// TIA Portal V20 export
DATA_BLOCK "InstCallEquipment"   // DB136
{ DB_Accessible_From_OPC_UA := 'FALSE' }
AUTHOR : ERsystem_FA2_DH. Kim
// stored: AssignedProDiagFB Unit1.Em2.ProDiag, DBAccessibleFromOPCUA false, DBAccessibleFromWebserver false, InstanceOfName Unit1.Em2.CallEquipment, InstanceOfType FB, Namespace Unit1.Em2
"Unit1.Em2.CallEquipment"
   // VAR_INPUT
   //    ZoneOperationEnable { ExternalWritable := 'False'} : "LWONIK_typeSafetyZoneManualOperation";
   // END_VAR
   // VAR_IN_OUT
   //    unitStatus : "LAF_typeUnitStatus";
   //    unitAlarmDB : "LAF_typeAlarms";
   //    emFeedback : "LUC_typeEmFeedback";
   // END_VAR
   // VAR
   //    instSequenceSemiAutoSplice { ExternalWritable := 'False'} : "Unit1.Em2.Sequence_1_SemiAutoSplice";
   //    instHomeJob1 { S7_SetPoint := 'True'} : "LAF_SelectJob";
   //    instJob2 { S7_SetPoint := 'True'} : "LAF_SelectJob";
   //    instJob3 { S7_SetPoint := 'True'} : "LAF_SelectJob";
   //    instJob4 { S7_SetPoint := 'True'} : "LAF_SelectJob";
   //    instJob5 { S7_SetPoint := 'True'} : "LAF_SelectJob";
   //    instJob6 { S7_SetPoint := 'True'} : "LAF_SelectJob";
   //    instJob7 { S7_SetPoint := 'True'} : "LAF_SelectJob";
   //    instJob8 { S7_SetPoint := 'True'} : "LAF_SelectJob";
   //    instJob9 { S7_SetPoint := 'True'} : "LAF_SelectJob";
   //    instJob10 { S7_SetPoint := 'True'} : "LAF_SelectJob";
   //    instJob11 { S7_SetPoint := 'True'} : "LAF_SelectJob";
   //    instJob12 { S7_SetPoint := 'True'} : "LAF_SelectJob";
   //    instJob13 { S7_SetPoint := 'True'} : "LAF_SelectJob";
   //    instJob14 { S7_SetPoint := 'True'} : "LAF_SelectJob";
   //    instJob15 { S7_SetPoint := 'True'} : "LAF_SelectJob";
   //    instJob16 { S7_SetPoint := 'True'} : "LAF_SelectJob";
   //    instJob17 { S7_SetPoint := 'True'} : "LAF_SelectJob";
   //    instJob18 { S7_SetPoint := 'True'} : "LAF_SelectJob";
   //    instJob19 { S7_SetPoint := 'True'} : "LAF_SelectJob";
   //    instJob20 { S7_SetPoint := 'True'} : "LAF_SelectJob";
   //    instJob21 { S7_SetPoint := 'True'} : "LAF_SelectJob";
   //    instJob22 { S7_SetPoint := 'True'} : "LAF_SelectJob";
   //    instJob23 { S7_SetPoint := 'True'} : "LAF_SelectJob";
   //    instJob24 { S7_SetPoint := 'True'} : "LAF_SelectJob";
   //    instJob25 { S7_SetPoint := 'True'} : "LAF_SelectJob";
   //    instJob26 { S7_SetPoint := 'True'} : "LAF_SelectJob";
   //    instJob27 { S7_SetPoint := 'True'} : "LAF_SelectJob";
   //    instJob28 { S7_SetPoint := 'True'} : "LAF_SelectJob";
   //    instJob29 { S7_SetPoint := 'True'} : "LAF_SelectJob";
   //    instJob30 { S7_SetPoint := 'True'} : "LAF_SelectJob";
   //    instBtmSepaVaccumJob4 { S7_SetPoint := 'True'} : "LAF_SelectJob";
   //    instCuttingJob5 { S7_SetPoint := 'True'} : "LAF_SelectJob";
   //    instTopSepaTransferJob6 { S7_SetPoint := 'True'} : "LAF_SelectJob";
   //    instBtmSepaTransferJob7 { S7_SetPoint := 'True'} : "LAF_SelectJob";
   //    instSuctionPadDownJob8 { S7_SetPoint := 'True'} : "LAF_SelectJob";
   //    instTopSepaReMoveJob9 { S7_SetPoint := 'True'} : "LAF_SelectJob";
   //    instBtmSepaReMoveJob10 { S7_SetPoint := 'True'} : "LAF_SelectJob";
   //    instTopSpliceRoateJob11 { S7_SetPoint := 'True'} : "LAF_SelectJob";
   //    instBtmSpliceRoateJob12 { S7_SetPoint := 'True'} : "LAF_SelectJob";
   //    instTopTapingStartJob13 { S7_SetPoint := 'True'} : "LAF_SelectJob";
   //    instBtmTapingStartJob14 { S7_SetPoint := 'True'} : "LAF_SelectJob";
   //    instTapingFinishJob15 { S7_SetPoint := 'True'} : "LAF_SelectJob";
   //    instFullAutoSplicingJob30 { S7_SetPoint := 'True'} : "LAF_SelectJob";
   //    instIsLink { S7_SetPoint := 'True'} : "LAF_SelectJob";
   //    instcmSuctionPadTopUpDown { ExternalAccessible := 'False'; ExternalVisible := 'False'; ExternalWritable := 'False'; S7_SetPoint := 'True'} : "LBC_TwoWayActuatorCn";
   //    instcmSuctionPadBtmUpDown { ExternalAccessible := 'False'; ExternalVisible := 'False'; ExternalWritable := 'False'; S7_SetPoint := 'True'} : "LBC_TwoWayActuatorCn";
   //    instcmCutterUpDown { ExternalAccessible := 'False'; ExternalVisible := 'False'; ExternalWritable := 'False'; S7_SetPoint := 'True'} : "LBC_TwoWayActuatorCn";
   //    instcmTapeTopUpDown { ExternalAccessible := 'False'; ExternalVisible := 'False'; ExternalWritable := 'False'; S7_SetPoint := 'True'} : "LBC_TwoWayActuatorCn";
   //    instcmTapeBtmUpDown { ExternalAccessible := 'False'; ExternalVisible := 'False'; ExternalWritable := 'False'; S7_SetPoint := 'True'} : "LBC_TwoWayActuatorCn";
   //    instcmSpliceHeadRotateTopFwdBwd { ExternalAccessible := 'False'; ExternalVisible := 'False'; ExternalWritable := 'False'; S7_SetPoint := 'True'} : "LBC_TwoWayActuatorCn";
   //    instcmSpliceHeadRotateBtmFwdBwd { ExternalAccessible := 'False'; ExternalVisible := 'False'; ExternalWritable := 'False'; S7_SetPoint := 'True'} : "LBC_TwoWayActuatorCn";
   //    instcmSuctionPadTopLeftVaccum { ExternalAccessible := 'False'; ExternalVisible := 'False'; ExternalWritable := 'False'; S7_SetPoint := 'True'} : "LBC_TwoWayActuatorCn";
   //    instcmSuctionPadTopRightVaccum { ExternalAccessible := 'False'; ExternalVisible := 'False'; ExternalWritable := 'False'; S7_SetPoint := 'True'} : "LBC_TwoWayActuatorCn";
   //    instCmSuctionPadBtmLeftVaccum { ExternalAccessible := 'False'; ExternalVisible := 'False'; ExternalWritable := 'False'; S7_SetPoint := 'True'} : "LBC_TwoWayActuatorCn";
   //    instCmSuctionPadBtmRightVaccum { ExternalAccessible := 'False'; ExternalVisible := 'False'; ExternalWritable := 'False'; S7_SetPoint := 'True'} : "LBC_TwoWayActuatorCn";
   //    instCmSuctionPadTopTapeVaccum { ExternalAccessible := 'False'; ExternalVisible := 'False'; ExternalWritable := 'False'; S7_SetPoint := 'True'} : "LBC_TwoWayActuatorCn";
   //    instCmSuctionPadBtmTapeVaccum { ExternalAccessible := 'False'; ExternalVisible := 'False'; ExternalWritable := 'False'; S7_SetPoint := 'True'} : "LBC_TwoWayActuatorCn";
   //    instManageAlarms { ExternalWritable := 'False'} : "LAF_ManageAlarms";
   //    instEventsPFE : "Unit1.Em2.EventsPFE";
   //    statTonTime { ExternalAccessible := 'False'; ExternalVisible := 'False'; ExternalWritable := 'False'} : Array[0..1999] of TON_TIME;
   //    statTofTime { ExternalAccessible := 'False'; ExternalVisible := 'False'; ExternalWritable := 'False'} : Array[0..99] of TOF_TIME;
   //    statPulse { ExternalAccessible := 'False'; ExternalVisible := 'False'; ExternalWritable := 'False'} : Array[0..999] of Bool;
   //    statUnitStatus { ExternalWritable := 'False'} : "LAF_typeUnitStatus";
   //    statEnableManualCmds : Bool := TRUE;
   //    Scan_on { ExternalAccessible := 'False'; ExternalVisible := 'False'; ExternalWritable := 'False'} : Bool;
   //    "*** Interlock Actuator ******" { ExternalAccessible := 'False'; ExternalVisible := 'False'; ExternalWritable := 'False'; S7_SetPoint := 'True'} : Bool;
   //    "SuctionPadTopUpDown Home" { S7_SetPoint := 'True'} : "Cylinder.LER_Actuator";
   //    "SuctionPadTopUpDown Work" { S7_SetPoint := 'True'} : "Cylinder.LER_Actuator";
   //    "SuctionPadBtmUpDown Home" { S7_SetPoint := 'True'} : "Cylinder.LER_Actuator";
   //    "SuctionPadBtmUpDown Work" { S7_SetPoint := 'True'} : "Cylinder.LER_Actuator";
   //    "CutterUpDown Home" { S7_SetPoint := 'True'} : "Cylinder.LER_Actuator";
   //    "CutterUpDown Work" { S7_SetPoint := 'True'} : "Cylinder.LER_Actuator";
   //    "TapeTopUpDown Home" { S7_SetPoint := 'True'} : "Cylinder.LER_Actuator";
   //    "TapeTopUpDown Work" { S7_SetPoint := 'True'} : "Cylinder.LER_Actuator";
   //    "TapeBtmUpDown Home" { S7_SetPoint := 'True'} : "Cylinder.LER_Actuator";
   //    "TapeBtmUpDown Work" { S7_SetPoint := 'True'} : "Cylinder.LER_Actuator";
   //    "SpliceHeadRotateTopFwdBwd Home" { S7_SetPoint := 'True'} : "Cylinder.LER_Actuator";
   //    "SpliceHeadRotateTopFwdBwd Work" { S7_SetPoint := 'True'} : "Cylinder.LER_Actuator";
   //    "SpliceHeadRotateBtmFwdBwd Home" { S7_SetPoint := 'True'} : "Cylinder.LER_Actuator";
   //    "SpliceHeadRotateBtmFwdBwd Work" { S7_SetPoint := 'True'} : "Cylinder.LER_Actuator";
   //    Cylinder3 : "LER_CM_Name";
   //    Vaccum1 : "LER_CM_Name";
   //    Vaccum6 : "LER_CM_Name";
   //    Cylinder8 : "LER_CM_Name";
   //    citi_Ptrig : Array[0..20] of Bool;
   //    citiTon : Array[0..20] of TON_TIME;
   //    citi : Time;
   //    citiTest : Array[0..20] of Bool;
   // END_VAR
BEGIN
   ZoneOperationEnable.autoStartEnable := FALSE;
   ZoneOperationEnable.doorLockEnable := TRUE;
   ZoneOperationEnable.doorUnlockEnable := TRUE;
   ZoneOperationEnable.rc_AutoEnable := FALSE;
   ZoneOperationEnable.rc_RollChangeEnable := FALSE;
   ZoneOperationEnable.rc_DoorLockEnable := TRUE;
   ZoneOperationEnable.rc_DoorUnlockEnable := TRUE;
   ZoneOperationEnable.hmiOperationEnable := TRUE;
   ZoneOperationEnable.phmiOperationEnable := FALSE;
   instcmSuctionPadTopUpDown.enable := TRUE;
   instcmSuctionPadTopUpDown.parentReferenceDesignator := WSTRING#'U1.EM2 SemiAutoSplice';
   instcmSuctionPadTopUpDown.feedbackHomePos := TRUE;
   instcmSuctionPadTopUpDown.feedbackWorkPos := FALSE;
   instcmSuctionPadTopUpDown.enableManualCmds := TRUE;
   instcmSuctionPadTopUpDown.interlockWorkPos := TRUE;
   instcmSuctionPadTopUpDown.interlockHomePos := TRUE;
   instcmSuctionPadTopUpDown.goToHomePos := FALSE;
   instcmSuctionPadTopUpDown.goToWorkPos := FALSE;
   instcmSuctionPadTopUpDown.statProcessValues.enable := TRUE;
   instcmSuctionPadTopUpDown.statProcessValues.referenceDesignator := WSTRING#'U1.EM2 SemiAutoSplice.cmSuctionPadTopUpDown';
   instcmSuctionPadTopUpDown.statProcessValues.commandHomePos := FALSE;
   instcmSuctionPadTopUpDown.statProcessValues.commandWorkPos := FALSE;
   instcmSuctionPadTopUpDown.statProcessValues.goToHomePos := FALSE;
   instcmSuctionPadTopUpDown.statProcessValues.goToWorkPos := FALSE;
   instcmSuctionPadTopUpDown.statProcessValues.inHomePos := FALSE;
   instcmSuctionPadTopUpDown.statProcessValues.inWorkPos := FALSE;
   instcmSuctionPadTopUpDown.statProcessValues.reset := FALSE;
   instcmSuctionPadTopUpDown.statProcessValues.enableManualCmds := TRUE;
   instcmSuctionPadTopUpDown.statProcessValues.error := FALSE;
   instcmSuctionPadTopUpDown.statProcessValues.interlockHomePos := TRUE;
   instcmSuctionPadTopUpDown.statProcessValues.interlockWorkPos := TRUE;
   instcmSuctionPadTopUpDown.statProcessValues.status := 16#7003;
   instcmSuctionPadTopUpDown.statProcessValues.interlockWarningWorkPos := FALSE;
   instcmSuctionPadTopUpDown.statProcessValues.interlockWarningHomePos := FALSE;
   instcmSuctionPadTopUpDown.statCurrentInputs.commandHomePos := FALSE;
   instcmSuctionPadTopUpDown.statCurrentInputs.commandWorkPos := FALSE;
   instcmSuctionPadTopUpDown.statCurrentInputs.reset := FALSE;
   instcmSuctionPadTopUpDown.statPreviousInputs.commandHomePos := FALSE;
   instcmSuctionPadTopUpDown.statPreviousInputs.commandWorkPos := FALSE;
   instcmSuctionPadTopUpDown.statPreviousInputs.reset := FALSE;
   instcmSuctionPadTopUpDown.statCurrentInterface.commandHomePos := FALSE;
   instcmSuctionPadTopUpDown.statCurrentInterface.commandWorkPos := FALSE;
   instcmSuctionPadTopUpDown.statCurrentInterface.reset := FALSE;
   instcmSuctionPadTopUpDown.statPreviousInterface.commandHomePos := FALSE;
   instcmSuctionPadTopUpDown.statPreviousInterface.commandWorkPos := FALSE;
   instcmSuctionPadTopUpDown.statPreviousInterface.reset := FALSE;
   instcmSuctionPadTopUpDown.statEmptyDiagnostics.status := 16#0000;
   instcmSuctionPadTopUpDown.statEmptyDiagnostics.subfunctionStatus := 16#0000;
   instcmSuctionPadTopUpDown.statEmptyDiagnostics.stateNumber := 0;
   instcmSuctionPadTopUpDown.instTimerReachPos.PT := T#0MS;
   instcmSuctionPadTopUpDown.instTimerReachPos.IN := FALSE;
   instcmSuctionPadTopUpDown.instTimerLeavePos.PT := T#0MS;
   instcmSuctionPadTopUpDown.instTimerLeavePos.IN := FALSE;
   instcmSuctionPadTopUpDown.instTimerDiscrepancyCheck.PT := T#0MS;
   instcmSuctionPadTopUpDown.instTimerDiscrepancyCheck.IN := FALSE;
   instcmSuctionPadTopUpDown.statDisableAlarms := TRUE;
   instcmSuctionPadTopUpDown.statDiagnostics.status := 16#7003;
   instcmSuctionPadTopUpDown.statDiagnostics.subfunctionStatus := 16#0000;
   instcmSuctionPadTopUpDown.statDiagnostics.stateNumber := 0;
   instcmSuctionPadTopUpDown.statEnablePrevious := TRUE;
   instcmSuctionPadTopUpDown.statFirstCall := FALSE;
   instcmSuctionPadTopUpDown.statResetPrevious := FALSE;
   instcmSuctionPadTopUpDown.statValid := TRUE;
   instcmSuctionPadTopUpDown.statBusy := TRUE;
   instcmSuctionPadTopUpDown.statError := FALSE;
   instcmSuctionPadTopUpDown.statInterlockWorkOff := FALSE;
   instcmSuctionPadTopUpDown.statInterlockHomeOff := FALSE;
   instcmSuctionPadTopUpDown.statFbState := 50;
   instcmSuctionPadTopUpDown.statFbStatePrevious := 50;
   instcmSuctionPadTopUpDown.statErrorUserCleared := FALSE;
   instcmSuctionPadTopUpDown.statErrorAutoCleared := FALSE;
   instcmSuctionPadTopUpDown.statErrorState := 16#0000;
   instcmSuctionPadTopUpDown.statDisablingCompleted := FALSE;
   instcmSuctionPadTopUpDown.statFeedbackHomePos := TRUE;
   instcmSuctionPadTopUpDown.statFeedbackWorkPos := FALSE;
   instcmSuctionPadBtmUpDown.enable := TRUE;
   instcmSuctionPadBtmUpDown.parentReferenceDesignator := WSTRING#'U1.EM2 SemiAutoSplice';
   instcmSuctionPadBtmUpDown.feedbackHomePos := TRUE;
   instcmSuctionPadBtmUpDown.feedbackWorkPos := FALSE;
   instcmSuctionPadBtmUpDown.enableManualCmds := TRUE;
   instcmSuctionPadBtmUpDown.interlockWorkPos := TRUE;
   instcmSuctionPadBtmUpDown.interlockHomePos := TRUE;
   instcmSuctionPadBtmUpDown.goToHomePos := FALSE;
   instcmSuctionPadBtmUpDown.goToWorkPos := FALSE;
   instcmSuctionPadBtmUpDown.statProcessValues.enable := TRUE;
   instcmSuctionPadBtmUpDown.statProcessValues.referenceDesignator := WSTRING#'U1.EM2 SemiAutoSplice.cmSuctionPadBtmUpDown';
   instcmSuctionPadBtmUpDown.statProcessValues.commandHomePos := FALSE;
   instcmSuctionPadBtmUpDown.statProcessValues.commandWorkPos := FALSE;
   instcmSuctionPadBtmUpDown.statProcessValues.goToHomePos := FALSE;
   instcmSuctionPadBtmUpDown.statProcessValues.goToWorkPos := FALSE;
   instcmSuctionPadBtmUpDown.statProcessValues.inHomePos := TRUE;
   instcmSuctionPadBtmUpDown.statProcessValues.inWorkPos := FALSE;
   instcmSuctionPadBtmUpDown.statProcessValues.reset := FALSE;
   instcmSuctionPadBtmUpDown.statProcessValues.enableManualCmds := TRUE;
   instcmSuctionPadBtmUpDown.statProcessValues.error := FALSE;
   instcmSuctionPadBtmUpDown.statProcessValues.interlockHomePos := TRUE;
   instcmSuctionPadBtmUpDown.statProcessValues.interlockWorkPos := TRUE;
   instcmSuctionPadBtmUpDown.statProcessValues.status := 16#7003;
   instcmSuctionPadBtmUpDown.statProcessValues.interlockWarningWorkPos := FALSE;
   instcmSuctionPadBtmUpDown.statProcessValues.interlockWarningHomePos := FALSE;
   instcmSuctionPadBtmUpDown.statCurrentInputs.commandHomePos := FALSE;
   instcmSuctionPadBtmUpDown.statCurrentInputs.commandWorkPos := FALSE;
   instcmSuctionPadBtmUpDown.statCurrentInputs.reset := FALSE;
   instcmSuctionPadBtmUpDown.statPreviousInputs.commandHomePos := FALSE;
   instcmSuctionPadBtmUpDown.statPreviousInputs.commandWorkPos := FALSE;
   instcmSuctionPadBtmUpDown.statPreviousInputs.reset := FALSE;
   instcmSuctionPadBtmUpDown.statCurrentInterface.commandHomePos := FALSE;
   instcmSuctionPadBtmUpDown.statCurrentInterface.commandWorkPos := FALSE;
   instcmSuctionPadBtmUpDown.statCurrentInterface.reset := FALSE;
   instcmSuctionPadBtmUpDown.statPreviousInterface.commandHomePos := FALSE;
   instcmSuctionPadBtmUpDown.statPreviousInterface.commandWorkPos := FALSE;
   instcmSuctionPadBtmUpDown.statPreviousInterface.reset := FALSE;
   instcmSuctionPadBtmUpDown.statEmptyDiagnostics.status := 16#0000;
   instcmSuctionPadBtmUpDown.statEmptyDiagnostics.subfunctionStatus := 16#0000;
   instcmSuctionPadBtmUpDown.statEmptyDiagnostics.stateNumber := 0;
   instcmSuctionPadBtmUpDown.instTimerReachPos.PT := T#0MS;
   instcmSuctionPadBtmUpDown.instTimerReachPos.IN := FALSE;
   instcmSuctionPadBtmUpDown.instTimerLeavePos.PT := T#0MS;
   instcmSuctionPadBtmUpDown.instTimerLeavePos.IN := FALSE;
   instcmSuctionPadBtmUpDown.instTimerDiscrepancyCheck.PT := T#0MS;
   instcmSuctionPadBtmUpDown.instTimerDiscrepancyCheck.IN := FALSE;
   instcmSuctionPadBtmUpDown.statDisableAlarms := TRUE;
   instcmSuctionPadBtmUpDown.statDiagnostics.status := 16#7003;
   instcmSuctionPadBtmUpDown.statDiagnostics.subfunctionStatus := 16#0000;
   instcmSuctionPadBtmUpDown.statDiagnostics.stateNumber := 0;
   instcmSuctionPadBtmUpDown.statEnablePrevious := TRUE;
   instcmSuctionPadBtmUpDown.statFirstCall := FALSE;
   instcmSuctionPadBtmUpDown.statResetPrevious := FALSE;
   instcmSuctionPadBtmUpDown.statValid := TRUE;
   instcmSuctionPadBtmUpDown.statBusy := TRUE;
   instcmSuctionPadBtmUpDown.statError := FALSE;
   instcmSuctionPadBtmUpDown.statInterlockWorkOff := FALSE;
   instcmSuctionPadBtmUpDown.statInterlockHomeOff := FALSE;
   instcmSuctionPadBtmUpDown.statFbState := 50;
   instcmSuctionPadBtmUpDown.statFbStatePrevious := 50;
   instcmSuctionPadBtmUpDown.statErrorUserCleared := FALSE;
   instcmSuctionPadBtmUpDown.statErrorAutoCleared := FALSE;
   instcmSuctionPadBtmUpDown.statErrorState := 16#0000;
   instcmSuctionPadBtmUpDown.statDisablingCompleted := FALSE;
   instcmSuctionPadBtmUpDown.statFeedbackHomePos := TRUE;
   instcmSuctionPadBtmUpDown.statFeedbackWorkPos := FALSE;
   instcmCutterUpDown.enable := TRUE;
   instcmCutterUpDown.parentReferenceDesignator := WSTRING#'U1.EM2 SemiAutoSplice';
   instcmCutterUpDown.feedbackHomePos := TRUE;
   instcmCutterUpDown.feedbackWorkPos := FALSE;
   instcmCutterUpDown.enableManualCmds := TRUE;
   instcmCutterUpDown.interlockWorkPos := FALSE;
   instcmCutterUpDown.interlockHomePos := TRUE;
   instcmCutterUpDown.goToHomePos := FALSE;
   instcmCutterUpDown.goToWorkPos := FALSE;
   instcmCutterUpDown.statProcessValues.enable := TRUE;
   instcmCutterUpDown.statProcessValues.referenceDesignator := WSTRING#'U1.EM2 SemiAutoSplice.cmCutterUpDown';
   instcmCutterUpDown.statProcessValues.commandHomePos := FALSE;
   instcmCutterUpDown.statProcessValues.commandWorkPos := FALSE;
   instcmCutterUpDown.statProcessValues.goToHomePos := FALSE;
   instcmCutterUpDown.statProcessValues.goToWorkPos := FALSE;
   instcmCutterUpDown.statProcessValues.inHomePos := TRUE;
   instcmCutterUpDown.statProcessValues.inWorkPos := FALSE;
   instcmCutterUpDown.statProcessValues.reset := FALSE;
   instcmCutterUpDown.statProcessValues.enableManualCmds := TRUE;
   instcmCutterUpDown.statProcessValues.error := FALSE;
   instcmCutterUpDown.statProcessValues.interlockHomePos := TRUE;
   instcmCutterUpDown.statProcessValues.interlockWorkPos := FALSE;
   instcmCutterUpDown.statProcessValues.status := 16#7101;
   instcmCutterUpDown.statProcessValues.interlockWarningWorkPos := FALSE;
   instcmCutterUpDown.statProcessValues.interlockWarningHomePos := FALSE;
   instcmCutterUpDown.statCurrentInputs.commandHomePos := FALSE;
   instcmCutterUpDown.statCurrentInputs.commandWorkPos := FALSE;
   instcmCutterUpDown.statCurrentInputs.reset := FALSE;
   instcmCutterUpDown.statPreviousInputs.commandHomePos := FALSE;
   instcmCutterUpDown.statPreviousInputs.commandWorkPos := FALSE;
   instcmCutterUpDown.statPreviousInputs.reset := FALSE;
   instcmCutterUpDown.statCurrentInterface.commandHomePos := FALSE;
   instcmCutterUpDown.statCurrentInterface.commandWorkPos := FALSE;
   instcmCutterUpDown.statCurrentInterface.reset := FALSE;
   instcmCutterUpDown.statPreviousInterface.commandHomePos := FALSE;
   instcmCutterUpDown.statPreviousInterface.commandWorkPos := FALSE;
   instcmCutterUpDown.statPreviousInterface.reset := FALSE;
   instcmCutterUpDown.statEmptyDiagnostics.status := 16#0000;
   instcmCutterUpDown.statEmptyDiagnostics.subfunctionStatus := 16#0000;
   instcmCutterUpDown.statEmptyDiagnostics.stateNumber := 0;
   instcmCutterUpDown.instTimerReachPos.PT := T#0MS;
   instcmCutterUpDown.instTimerReachPos.IN := FALSE;
   instcmCutterUpDown.instTimerLeavePos.PT := T#0MS;
   instcmCutterUpDown.instTimerLeavePos.IN := FALSE;
   instcmCutterUpDown.instTimerDiscrepancyCheck.PT := T#0MS;
   instcmCutterUpDown.instTimerDiscrepancyCheck.IN := FALSE;
   instcmCutterUpDown.statDisableAlarms := TRUE;
   instcmCutterUpDown.statDiagnostics.status := 16#7003;
   instcmCutterUpDown.statDiagnostics.subfunctionStatus := 16#0000;
   instcmCutterUpDown.statDiagnostics.stateNumber := 0;
   instcmCutterUpDown.statEnablePrevious := TRUE;
   instcmCutterUpDown.statFirstCall := FALSE;
   instcmCutterUpDown.statResetPrevious := FALSE;
   instcmCutterUpDown.statValid := TRUE;
   instcmCutterUpDown.statBusy := TRUE;
   instcmCutterUpDown.statError := FALSE;
   instcmCutterUpDown.statInterlockWorkOff := FALSE;
   instcmCutterUpDown.statInterlockHomeOff := FALSE;
   instcmCutterUpDown.statFbState := 50;
   instcmCutterUpDown.statFbStatePrevious := 50;
   instcmCutterUpDown.statErrorUserCleared := FALSE;
   instcmCutterUpDown.statErrorAutoCleared := FALSE;
   instcmCutterUpDown.statErrorState := 16#0000;
   instcmCutterUpDown.statDisablingCompleted := FALSE;
   instcmCutterUpDown.statFeedbackHomePos := TRUE;
   instcmCutterUpDown.statFeedbackWorkPos := FALSE;
   instcmTapeTopUpDown.enable := TRUE;
   instcmTapeTopUpDown.parentReferenceDesignator := WSTRING#'U1.EM2 SemiAutoSplice';
   instcmTapeTopUpDown.feedbackHomePos := FALSE;
   instcmTapeTopUpDown.feedbackWorkPos := TRUE;
   instcmTapeTopUpDown.enableManualCmds := TRUE;
   instcmTapeTopUpDown.interlockWorkPos := FALSE;
   instcmTapeTopUpDown.interlockHomePos := TRUE;
   instcmTapeTopUpDown.goToHomePos := FALSE;
   instcmTapeTopUpDown.goToWorkPos := FALSE;
   instcmTapeTopUpDown.statProcessValues.enable := TRUE;
   instcmTapeTopUpDown.statProcessValues.referenceDesignator := WSTRING#'U1.EM2 SemiAutoSplice.cmTapeTopUpDown';
   instcmTapeTopUpDown.statProcessValues.commandHomePos := FALSE;
   instcmTapeTopUpDown.statProcessValues.commandWorkPos := FALSE;
   instcmTapeTopUpDown.statProcessValues.goToHomePos := FALSE;
   instcmTapeTopUpDown.statProcessValues.goToWorkPos := FALSE;
   instcmTapeTopUpDown.statProcessValues.inHomePos := FALSE;
   instcmTapeTopUpDown.statProcessValues.inWorkPos := FALSE;
   instcmTapeTopUpDown.statProcessValues.reset := FALSE;
   instcmTapeTopUpDown.statProcessValues.enableManualCmds := TRUE;
   instcmTapeTopUpDown.statProcessValues.error := FALSE;
   instcmTapeTopUpDown.statProcessValues.interlockHomePos := TRUE;
   instcmTapeTopUpDown.statProcessValues.interlockWorkPos := FALSE;
   instcmTapeTopUpDown.statProcessValues.status := 16#7101;
   instcmTapeTopUpDown.statProcessValues.interlockWarningWorkPos := FALSE;
   instcmTapeTopUpDown.statProcessValues.interlockWarningHomePos := FALSE;
   instcmTapeTopUpDown.statCurrentInputs.commandHomePos := FALSE;
   instcmTapeTopUpDown.statCurrentInputs.commandWorkPos := FALSE;
   instcmTapeTopUpDown.statCurrentInputs.reset := FALSE;
   instcmTapeTopUpDown.statPreviousInputs.commandHomePos := FALSE;
   instcmTapeTopUpDown.statPreviousInputs.commandWorkPos := FALSE;
   instcmTapeTopUpDown.statPreviousInputs.reset := FALSE;
   instcmTapeTopUpDown.statCurrentInterface.commandHomePos := FALSE;
   instcmTapeTopUpDown.statCurrentInterface.commandWorkPos := FALSE;
   instcmTapeTopUpDown.statCurrentInterface.reset := FALSE;
   instcmTapeTopUpDown.statPreviousInterface.commandHomePos := FALSE;
   instcmTapeTopUpDown.statPreviousInterface.commandWorkPos := FALSE;
   instcmTapeTopUpDown.statPreviousInterface.reset := FALSE;
   instcmTapeTopUpDown.statEmptyDiagnostics.status := 16#0000;
   instcmTapeTopUpDown.statEmptyDiagnostics.subfunctionStatus := 16#0000;
   instcmTapeTopUpDown.statEmptyDiagnostics.stateNumber := 0;
   instcmTapeTopUpDown.instTimerReachPos.PT := T#0MS;
   instcmTapeTopUpDown.instTimerReachPos.IN := FALSE;
   instcmTapeTopUpDown.instTimerLeavePos.PT := T#0MS;
   instcmTapeTopUpDown.instTimerLeavePos.IN := FALSE;
   instcmTapeTopUpDown.instTimerDiscrepancyCheck.PT := T#0MS;
   instcmTapeTopUpDown.instTimerDiscrepancyCheck.IN := FALSE;
   instcmTapeTopUpDown.statDisableAlarms := TRUE;
   instcmTapeTopUpDown.statDiagnostics.status := 16#7003;
   instcmTapeTopUpDown.statDiagnostics.subfunctionStatus := 16#0000;
   instcmTapeTopUpDown.statDiagnostics.stateNumber := 0;
   instcmTapeTopUpDown.statEnablePrevious := TRUE;
   instcmTapeTopUpDown.statFirstCall := FALSE;
   instcmTapeTopUpDown.statResetPrevious := FALSE;
   instcmTapeTopUpDown.statValid := TRUE;
   instcmTapeTopUpDown.statBusy := TRUE;
   instcmTapeTopUpDown.statError := FALSE;
   instcmTapeTopUpDown.statInterlockWorkOff := FALSE;
   instcmTapeTopUpDown.statInterlockHomeOff := FALSE;
   instcmTapeTopUpDown.statFbState := 50;
   instcmTapeTopUpDown.statFbStatePrevious := 50;
   instcmTapeTopUpDown.statErrorUserCleared := FALSE;
   instcmTapeTopUpDown.statErrorAutoCleared := FALSE;
   instcmTapeTopUpDown.statErrorState := 16#0000;
   instcmTapeTopUpDown.statDisablingCompleted := FALSE;
   instcmTapeTopUpDown.statFeedbackHomePos := FALSE;
   instcmTapeTopUpDown.statFeedbackWorkPos := TRUE;
   instcmTapeBtmUpDown.enable := TRUE;
   instcmTapeBtmUpDown.parentReferenceDesignator := WSTRING#'U1.EM2 SemiAutoSplice';
   instcmTapeBtmUpDown.feedbackHomePos := TRUE;
   instcmTapeBtmUpDown.feedbackWorkPos := FALSE;
   instcmTapeBtmUpDown.enableManualCmds := TRUE;
   instcmTapeBtmUpDown.interlockWorkPos := FALSE;
   instcmTapeBtmUpDown.interlockHomePos := TRUE;
   instcmTapeBtmUpDown.goToHomePos := FALSE;
   instcmTapeBtmUpDown.goToWorkPos := FALSE;
   instcmTapeBtmUpDown.statProcessValues.enable := TRUE;
   instcmTapeBtmUpDown.statProcessValues.referenceDesignator := WSTRING#'U1.EM2 SemiAutoSplice.cmTapeBtmUpDown';
   instcmTapeBtmUpDown.statProcessValues.commandHomePos := FALSE;
   instcmTapeBtmUpDown.statProcessValues.commandWorkPos := FALSE;
   instcmTapeBtmUpDown.statProcessValues.goToHomePos := FALSE;
   instcmTapeBtmUpDown.statProcessValues.goToWorkPos := FALSE;
   instcmTapeBtmUpDown.statProcessValues.inHomePos := TRUE;
   instcmTapeBtmUpDown.statProcessValues.inWorkPos := FALSE;
   instcmTapeBtmUpDown.statProcessValues.reset := FALSE;
   instcmTapeBtmUpDown.statProcessValues.enableManualCmds := TRUE;
   instcmTapeBtmUpDown.statProcessValues.error := FALSE;
   instcmTapeBtmUpDown.statProcessValues.interlockHomePos := TRUE;
   instcmTapeBtmUpDown.statProcessValues.interlockWorkPos := FALSE;
   instcmTapeBtmUpDown.statProcessValues.status := 16#7101;
   instcmTapeBtmUpDown.statProcessValues.interlockWarningWorkPos := FALSE;
   instcmTapeBtmUpDown.statProcessValues.interlockWarningHomePos := FALSE;
   instcmTapeBtmUpDown.statCurrentInputs.commandHomePos := FALSE;
   instcmTapeBtmUpDown.statCurrentInputs.commandWorkPos := FALSE;
   instcmTapeBtmUpDown.statCurrentInputs.reset := FALSE;
   instcmTapeBtmUpDown.statPreviousInputs.commandHomePos := FALSE;
   instcmTapeBtmUpDown.statPreviousInputs.commandWorkPos := FALSE;
   instcmTapeBtmUpDown.statPreviousInputs.reset := FALSE;
   instcmTapeBtmUpDown.statCurrentInterface.commandHomePos := FALSE;
   instcmTapeBtmUpDown.statCurrentInterface.commandWorkPos := FALSE;
   instcmTapeBtmUpDown.statCurrentInterface.reset := FALSE;
   instcmTapeBtmUpDown.statPreviousInterface.commandHomePos := FALSE;
   instcmTapeBtmUpDown.statPreviousInterface.commandWorkPos := FALSE;
   instcmTapeBtmUpDown.statPreviousInterface.reset := FALSE;
   instcmTapeBtmUpDown.statEmptyDiagnostics.status := 16#0000;
   instcmTapeBtmUpDown.statEmptyDiagnostics.subfunctionStatus := 16#0000;
   instcmTapeBtmUpDown.statEmptyDiagnostics.stateNumber := 0;
   instcmTapeBtmUpDown.instTimerReachPos.PT := T#0MS;
   instcmTapeBtmUpDown.instTimerReachPos.IN := FALSE;
   instcmTapeBtmUpDown.instTimerLeavePos.PT := T#0MS;
   instcmTapeBtmUpDown.instTimerLeavePos.IN := FALSE;
   instcmTapeBtmUpDown.instTimerDiscrepancyCheck.PT := T#0MS;
   instcmTapeBtmUpDown.instTimerDiscrepancyCheck.IN := FALSE;
   instcmTapeBtmUpDown.statDisableAlarms := TRUE;
   instcmTapeBtmUpDown.statDiagnostics.status := 16#7003;
   instcmTapeBtmUpDown.statDiagnostics.subfunctionStatus := 16#0000;
   instcmTapeBtmUpDown.statDiagnostics.stateNumber := 0;
   instcmTapeBtmUpDown.statEnablePrevious := TRUE;
   instcmTapeBtmUpDown.statFirstCall := FALSE;
   instcmTapeBtmUpDown.statResetPrevious := FALSE;
   instcmTapeBtmUpDown.statValid := TRUE;
   instcmTapeBtmUpDown.statBusy := TRUE;
   instcmTapeBtmUpDown.statError := FALSE;
   instcmTapeBtmUpDown.statInterlockWorkOff := FALSE;
   instcmTapeBtmUpDown.statInterlockHomeOff := FALSE;
   instcmTapeBtmUpDown.statFbState := 50;
   instcmTapeBtmUpDown.statFbStatePrevious := 50;
   instcmTapeBtmUpDown.statErrorUserCleared := FALSE;
   instcmTapeBtmUpDown.statErrorAutoCleared := FALSE;
   instcmTapeBtmUpDown.statErrorState := 16#0000;
   instcmTapeBtmUpDown.statDisablingCompleted := FALSE;
   instcmTapeBtmUpDown.statFeedbackHomePos := TRUE;
   instcmTapeBtmUpDown.statFeedbackWorkPos := FALSE;
   instcmSpliceHeadRotateTopFwdBwd.enable := TRUE;
   instcmSpliceHeadRotateTopFwdBwd.parentReferenceDesignator := WSTRING#'U1.EM2 SemiAutoSplice';
   instcmSpliceHeadRotateTopFwdBwd.feedbackHomePos := TRUE;
   instcmSpliceHeadRotateTopFwdBwd.feedbackWorkPos := FALSE;
   instcmSpliceHeadRotateTopFwdBwd.enableManualCmds := TRUE;
   instcmSpliceHeadRotateTopFwdBwd.interlockWorkPos := FALSE;
   instcmSpliceHeadRotateTopFwdBwd.interlockHomePos := FALSE;
   instcmSpliceHeadRotateTopFwdBwd.goToHomePos := FALSE;
   instcmSpliceHeadRotateTopFwdBwd.goToWorkPos := FALSE;
   instcmSpliceHeadRotateTopFwdBwd.statProcessValues.enable := TRUE;
   instcmSpliceHeadRotateTopFwdBwd.statProcessValues.referenceDesignator := WSTRING#'U1.EM2 SemiAutoSplice.cmSpliceRotateTopFwdBwd';
   instcmSpliceHeadRotateTopFwdBwd.statProcessValues.commandHomePos := FALSE;
   instcmSpliceHeadRotateTopFwdBwd.statProcessValues.commandWorkPos := FALSE;
   instcmSpliceHeadRotateTopFwdBwd.statProcessValues.goToHomePos := FALSE;
   instcmSpliceHeadRotateTopFwdBwd.statProcessValues.goToWorkPos := FALSE;
   instcmSpliceHeadRotateTopFwdBwd.statProcessValues.inHomePos := TRUE;
   instcmSpliceHeadRotateTopFwdBwd.statProcessValues.inWorkPos := FALSE;
   instcmSpliceHeadRotateTopFwdBwd.statProcessValues.reset := FALSE;
   instcmSpliceHeadRotateTopFwdBwd.statProcessValues.enableManualCmds := TRUE;
   instcmSpliceHeadRotateTopFwdBwd.statProcessValues.error := FALSE;
   instcmSpliceHeadRotateTopFwdBwd.statProcessValues.interlockHomePos := FALSE;
   instcmSpliceHeadRotateTopFwdBwd.statProcessValues.interlockWorkPos := FALSE;
   instcmSpliceHeadRotateTopFwdBwd.statProcessValues.status := 16#7100;
   instcmSpliceHeadRotateTopFwdBwd.statProcessValues.interlockWarningWorkPos := FALSE;
   instcmSpliceHeadRotateTopFwdBwd.statProcessValues.interlockWarningHomePos := FALSE;
   instcmSpliceHeadRotateTopFwdBwd.statCurrentInputs.commandHomePos := FALSE;
   instcmSpliceHeadRotateTopFwdBwd.statCurrentInputs.commandWorkPos := FALSE;
   instcmSpliceHeadRotateTopFwdBwd.statCurrentInputs.reset := FALSE;
   instcmSpliceHeadRotateTopFwdBwd.statPreviousInputs.commandHomePos := FALSE;
   instcmSpliceHeadRotateTopFwdBwd.statPreviousInputs.commandWorkPos := FALSE;
   instcmSpliceHeadRotateTopFwdBwd.statPreviousInputs.reset := FALSE;
   instcmSpliceHeadRotateTopFwdBwd.statCurrentInterface.commandHomePos := FALSE;
   instcmSpliceHeadRotateTopFwdBwd.statCurrentInterface.commandWorkPos := FALSE;
   instcmSpliceHeadRotateTopFwdBwd.statCurrentInterface.reset := FALSE;
   instcmSpliceHeadRotateTopFwdBwd.statPreviousInterface.commandHomePos := FALSE;
   instcmSpliceHeadRotateTopFwdBwd.statPreviousInterface.commandWorkPos := FALSE;
   instcmSpliceHeadRotateTopFwdBwd.statPreviousInterface.reset := FALSE;
   instcmSpliceHeadRotateTopFwdBwd.statEmptyDiagnostics.status := 16#0000;
   instcmSpliceHeadRotateTopFwdBwd.statEmptyDiagnostics.subfunctionStatus := 16#0000;
   instcmSpliceHeadRotateTopFwdBwd.statEmptyDiagnostics.stateNumber := 0;
   instcmSpliceHeadRotateTopFwdBwd.instTimerReachPos.PT := T#0MS;
   instcmSpliceHeadRotateTopFwdBwd.instTimerReachPos.IN := FALSE;
   instcmSpliceHeadRotateTopFwdBwd.instTimerLeavePos.PT := T#0MS;
   instcmSpliceHeadRotateTopFwdBwd.instTimerLeavePos.IN := FALSE;
   instcmSpliceHeadRotateTopFwdBwd.instTimerDiscrepancyCheck.PT := T#0MS;
   instcmSpliceHeadRotateTopFwdBwd.instTimerDiscrepancyCheck.IN := FALSE;
   instcmSpliceHeadRotateTopFwdBwd.statDisableAlarms := TRUE;
   instcmSpliceHeadRotateTopFwdBwd.statDiagnostics.status := 16#7003;
   instcmSpliceHeadRotateTopFwdBwd.statDiagnostics.subfunctionStatus := 16#0000;
   instcmSpliceHeadRotateTopFwdBwd.statDiagnostics.stateNumber := 0;
   instcmSpliceHeadRotateTopFwdBwd.statEnablePrevious := TRUE;
   instcmSpliceHeadRotateTopFwdBwd.statFirstCall := FALSE;
   instcmSpliceHeadRotateTopFwdBwd.statResetPrevious := FALSE;
   instcmSpliceHeadRotateTopFwdBwd.statValid := TRUE;
   instcmSpliceHeadRotateTopFwdBwd.statBusy := TRUE;
   instcmSpliceHeadRotateTopFwdBwd.statError := FALSE;
   instcmSpliceHeadRotateTopFwdBwd.statInterlockWorkOff := FALSE;
   instcmSpliceHeadRotateTopFwdBwd.statInterlockHomeOff := FALSE;
   instcmSpliceHeadRotateTopFwdBwd.statFbState := 50;
   instcmSpliceHeadRotateTopFwdBwd.statFbStatePrevious := 50;
   instcmSpliceHeadRotateTopFwdBwd.statErrorUserCleared := FALSE;
   instcmSpliceHeadRotateTopFwdBwd.statErrorAutoCleared := FALSE;
   instcmSpliceHeadRotateTopFwdBwd.statErrorState := 16#0000;
   instcmSpliceHeadRotateTopFwdBwd.statDisablingCompleted := FALSE;
   instcmSpliceHeadRotateTopFwdBwd.statFeedbackHomePos := TRUE;
   instcmSpliceHeadRotateTopFwdBwd.statFeedbackWorkPos := FALSE;
   instcmSpliceHeadRotateBtmFwdBwd.enable := TRUE;
   instcmSpliceHeadRotateBtmFwdBwd.parentReferenceDesignator := WSTRING#'U1.EM2 SemiAutoSplice';
   instcmSpliceHeadRotateBtmFwdBwd.feedbackHomePos := TRUE;
   instcmSpliceHeadRotateBtmFwdBwd.feedbackWorkPos := FALSE;
   instcmSpliceHeadRotateBtmFwdBwd.enableManualCmds := TRUE;
   instcmSpliceHeadRotateBtmFwdBwd.interlockWorkPos := FALSE;
   instcmSpliceHeadRotateBtmFwdBwd.interlockHomePos := FALSE;
   instcmSpliceHeadRotateBtmFwdBwd.goToHomePos := FALSE;
   instcmSpliceHeadRotateBtmFwdBwd.goToWorkPos := FALSE;
   instcmSpliceHeadRotateBtmFwdBwd.statProcessValues.enable := TRUE;
   instcmSpliceHeadRotateBtmFwdBwd.statProcessValues.referenceDesignator := WSTRING#'U1.EM2 SemiAutoSplice.cmSpliceRotateBtmFwdBwd';
   instcmSpliceHeadRotateBtmFwdBwd.statProcessValues.commandHomePos := FALSE;
   instcmSpliceHeadRotateBtmFwdBwd.statProcessValues.commandWorkPos := FALSE;
   instcmSpliceHeadRotateBtmFwdBwd.statProcessValues.goToHomePos := FALSE;
   instcmSpliceHeadRotateBtmFwdBwd.statProcessValues.goToWorkPos := FALSE;
   instcmSpliceHeadRotateBtmFwdBwd.statProcessValues.inHomePos := TRUE;
   instcmSpliceHeadRotateBtmFwdBwd.statProcessValues.inWorkPos := FALSE;
   instcmSpliceHeadRotateBtmFwdBwd.statProcessValues.reset := FALSE;
   instcmSpliceHeadRotateBtmFwdBwd.statProcessValues.enableManualCmds := TRUE;
   instcmSpliceHeadRotateBtmFwdBwd.statProcessValues.error := FALSE;
   instcmSpliceHeadRotateBtmFwdBwd.statProcessValues.interlockHomePos := FALSE;
   instcmSpliceHeadRotateBtmFwdBwd.statProcessValues.interlockWorkPos := FALSE;
   instcmSpliceHeadRotateBtmFwdBwd.statProcessValues.status := 16#7100;
   instcmSpliceHeadRotateBtmFwdBwd.statProcessValues.interlockWarningWorkPos := FALSE;
   instcmSpliceHeadRotateBtmFwdBwd.statProcessValues.interlockWarningHomePos := FALSE;
   instcmSpliceHeadRotateBtmFwdBwd.statCurrentInputs.commandHomePos := FALSE;
   instcmSpliceHeadRotateBtmFwdBwd.statCurrentInputs.commandWorkPos := FALSE;
   instcmSpliceHeadRotateBtmFwdBwd.statCurrentInputs.reset := FALSE;
   instcmSpliceHeadRotateBtmFwdBwd.statPreviousInputs.commandHomePos := FALSE;
   instcmSpliceHeadRotateBtmFwdBwd.statPreviousInputs.commandWorkPos := FALSE;
   instcmSpliceHeadRotateBtmFwdBwd.statPreviousInputs.reset := FALSE;
   instcmSpliceHeadRotateBtmFwdBwd.statCurrentInterface.commandHomePos := FALSE;
   instcmSpliceHeadRotateBtmFwdBwd.statCurrentInterface.commandWorkPos := FALSE;
   instcmSpliceHeadRotateBtmFwdBwd.statCurrentInterface.reset := FALSE;
   instcmSpliceHeadRotateBtmFwdBwd.statPreviousInterface.commandHomePos := FALSE;
   instcmSpliceHeadRotateBtmFwdBwd.statPreviousInterface.commandWorkPos := FALSE;
   instcmSpliceHeadRotateBtmFwdBwd.statPreviousInterface.reset := FALSE;
   instcmSpliceHeadRotateBtmFwdBwd.statEmptyDiagnostics.status := 16#0000;
   instcmSpliceHeadRotateBtmFwdBwd.statEmptyDiagnostics.subfunctionStatus := 16#0000;
   instcmSpliceHeadRotateBtmFwdBwd.statEmptyDiagnostics.stateNumber := 0;
   instcmSpliceHeadRotateBtmFwdBwd.instTimerReachPos.PT := T#0MS;
   instcmSpliceHeadRotateBtmFwdBwd.instTimerReachPos.IN := FALSE;
   instcmSpliceHeadRotateBtmFwdBwd.instTimerLeavePos.PT := T#0MS;
   instcmSpliceHeadRotateBtmFwdBwd.instTimerLeavePos.IN := FALSE;
   instcmSpliceHeadRotateBtmFwdBwd.instTimerDiscrepancyCheck.PT := T#0MS;
   instcmSpliceHeadRotateBtmFwdBwd.instTimerDiscrepancyCheck.IN := FALSE;
   instcmSpliceHeadRotateBtmFwdBwd.statDisableAlarms := TRUE;
   instcmSpliceHeadRotateBtmFwdBwd.statDiagnostics.status := 16#7003;
   instcmSpliceHeadRotateBtmFwdBwd.statDiagnostics.subfunctionStatus := 16#0000;
   instcmSpliceHeadRotateBtmFwdBwd.statDiagnostics.stateNumber := 0;
   instcmSpliceHeadRotateBtmFwdBwd.statEnablePrevious := TRUE;
   instcmSpliceHeadRotateBtmFwdBwd.statFirstCall := FALSE;
   instcmSpliceHeadRotateBtmFwdBwd.statResetPrevious := FALSE;
   instcmSpliceHeadRotateBtmFwdBwd.statValid := TRUE;
   instcmSpliceHeadRotateBtmFwdBwd.statBusy := TRUE;
   instcmSpliceHeadRotateBtmFwdBwd.statError := FALSE;
   instcmSpliceHeadRotateBtmFwdBwd.statInterlockWorkOff := FALSE;
   instcmSpliceHeadRotateBtmFwdBwd.statInterlockHomeOff := FALSE;
   instcmSpliceHeadRotateBtmFwdBwd.statFbState := 50;
   instcmSpliceHeadRotateBtmFwdBwd.statFbStatePrevious := 50;
   instcmSpliceHeadRotateBtmFwdBwd.statErrorUserCleared := FALSE;
   instcmSpliceHeadRotateBtmFwdBwd.statErrorAutoCleared := FALSE;
   instcmSpliceHeadRotateBtmFwdBwd.statErrorState := 16#0000;
   instcmSpliceHeadRotateBtmFwdBwd.statDisablingCompleted := FALSE;
   instcmSpliceHeadRotateBtmFwdBwd.statFeedbackHomePos := TRUE;
   instcmSpliceHeadRotateBtmFwdBwd.statFeedbackWorkPos := FALSE;
   instcmSuctionPadTopLeftVaccum.enable := TRUE;
   instcmSuctionPadTopLeftVaccum.parentReferenceDesignator := WSTRING#'U1.EM2 SemiAutoSplice';
   instcmSuctionPadTopLeftVaccum.feedbackHomePos := TRUE;
   instcmSuctionPadTopLeftVaccum.feedbackWorkPos := FALSE;
   instcmSuctionPadTopLeftVaccum.enableManualCmds := TRUE;
   instcmSuctionPadTopLeftVaccum.interlockWorkPos := TRUE;
   instcmSuctionPadTopLeftVaccum.interlockHomePos := TRUE;
   instcmSuctionPadTopLeftVaccum.goToHomePos := FALSE;
   instcmSuctionPadTopLeftVaccum.goToWorkPos := FALSE;
   instcmSuctionPadTopLeftVaccum.statProcessValues.enable := TRUE;
   instcmSuctionPadTopLeftVaccum.statProcessValues.referenceDesignator := WSTRING#'U1.EM2 SemiAutoSplice.cmSuctionPadTopLeftVac';
   instcmSuctionPadTopLeftVaccum.statProcessValues.commandHomePos := FALSE;
   instcmSuctionPadTopLeftVaccum.statProcessValues.commandWorkPos := FALSE;
   instcmSuctionPadTopLeftVaccum.statProcessValues.goToHomePos := FALSE;
   instcmSuctionPadTopLeftVaccum.statProcessValues.goToWorkPos := FALSE;
   instcmSuctionPadTopLeftVaccum.statProcessValues.inHomePos := TRUE;
   instcmSuctionPadTopLeftVaccum.statProcessValues.inWorkPos := FALSE;
   instcmSuctionPadTopLeftVaccum.statProcessValues.reset := FALSE;
   instcmSuctionPadTopLeftVaccum.statProcessValues.enableManualCmds := TRUE;
   instcmSuctionPadTopLeftVaccum.statProcessValues.error := FALSE;
   instcmSuctionPadTopLeftVaccum.statProcessValues.interlockHomePos := TRUE;
   instcmSuctionPadTopLeftVaccum.statProcessValues.interlockWorkPos := TRUE;
   instcmSuctionPadTopLeftVaccum.statProcessValues.status := 16#7003;
   instcmSuctionPadTopLeftVaccum.statProcessValues.interlockWarningWorkPos := FALSE;
   instcmSuctionPadTopLeftVaccum.statProcessValues.interlockWarningHomePos := FALSE;
   instcmSuctionPadTopLeftVaccum.statCurrentInputs.commandHomePos := FALSE;
   instcmSuctionPadTopLeftVaccum.statCurrentInputs.commandWorkPos := FALSE;
   instcmSuctionPadTopLeftVaccum.statCurrentInputs.reset := FALSE;
   instcmSuctionPadTopLeftVaccum.statPreviousInputs.commandHomePos := FALSE;
   instcmSuctionPadTopLeftVaccum.statPreviousInputs.commandWorkPos := FALSE;
   instcmSuctionPadTopLeftVaccum.statPreviousInputs.reset := FALSE;
   instcmSuctionPadTopLeftVaccum.statCurrentInterface.commandHomePos := FALSE;
   instcmSuctionPadTopLeftVaccum.statCurrentInterface.commandWorkPos := FALSE;
   instcmSuctionPadTopLeftVaccum.statCurrentInterface.reset := FALSE;
   instcmSuctionPadTopLeftVaccum.statPreviousInterface.commandHomePos := FALSE;
   instcmSuctionPadTopLeftVaccum.statPreviousInterface.commandWorkPos := FALSE;
   instcmSuctionPadTopLeftVaccum.statPreviousInterface.reset := FALSE;
   instcmSuctionPadTopLeftVaccum.statEmptyDiagnostics.status := 16#0000;
   instcmSuctionPadTopLeftVaccum.statEmptyDiagnostics.subfunctionStatus := 16#0000;
   instcmSuctionPadTopLeftVaccum.statEmptyDiagnostics.stateNumber := 0;
   instcmSuctionPadTopLeftVaccum.instTimerReachPos.PT := T#0MS;
   instcmSuctionPadTopLeftVaccum.instTimerReachPos.IN := FALSE;
   instcmSuctionPadTopLeftVaccum.instTimerLeavePos.PT := T#0MS;
   instcmSuctionPadTopLeftVaccum.instTimerLeavePos.IN := FALSE;
   instcmSuctionPadTopLeftVaccum.instTimerDiscrepancyCheck.PT := T#0MS;
   instcmSuctionPadTopLeftVaccum.instTimerDiscrepancyCheck.IN := FALSE;
   instcmSuctionPadTopLeftVaccum.statDisableAlarms := FALSE;
   instcmSuctionPadTopLeftVaccum.statDiagnostics.status := 16#7003;
   instcmSuctionPadTopLeftVaccum.statDiagnostics.subfunctionStatus := 16#0000;
   instcmSuctionPadTopLeftVaccum.statDiagnostics.stateNumber := 0;
   instcmSuctionPadTopLeftVaccum.statEnablePrevious := TRUE;
   instcmSuctionPadTopLeftVaccum.statFirstCall := FALSE;
   instcmSuctionPadTopLeftVaccum.statResetPrevious := FALSE;
   instcmSuctionPadTopLeftVaccum.statValid := TRUE;
   instcmSuctionPadTopLeftVaccum.statBusy := TRUE;
   instcmSuctionPadTopLeftVaccum.statError := FALSE;
   instcmSuctionPadTopLeftVaccum.statInterlockWorkOff := FALSE;
   instcmSuctionPadTopLeftVaccum.statInterlockHomeOff := FALSE;
   instcmSuctionPadTopLeftVaccum.statFbState := 50;
   instcmSuctionPadTopLeftVaccum.statFbStatePrevious := 50;
   instcmSuctionPadTopLeftVaccum.statErrorUserCleared := FALSE;
   instcmSuctionPadTopLeftVaccum.statErrorAutoCleared := FALSE;
   instcmSuctionPadTopLeftVaccum.statErrorState := 16#0000;
   instcmSuctionPadTopLeftVaccum.statDisablingCompleted := FALSE;
   instcmSuctionPadTopLeftVaccum.statFeedbackHomePos := TRUE;
   instcmSuctionPadTopLeftVaccum.statFeedbackWorkPos := FALSE;
   instcmSuctionPadTopRightVaccum.enable := TRUE;
   instcmSuctionPadTopRightVaccum.parentReferenceDesignator := WSTRING#'U1.EM2 SemiAutoSplice';
   instcmSuctionPadTopRightVaccum.feedbackHomePos := TRUE;
   instcmSuctionPadTopRightVaccum.feedbackWorkPos := FALSE;
   instcmSuctionPadTopRightVaccum.enableManualCmds := TRUE;
   instcmSuctionPadTopRightVaccum.interlockWorkPos := TRUE;
   instcmSuctionPadTopRightVaccum.interlockHomePos := TRUE;
   instcmSuctionPadTopRightVaccum.goToHomePos := FALSE;
   instcmSuctionPadTopRightVaccum.goToWorkPos := FALSE;
   instcmSuctionPadTopRightVaccum.statProcessValues.enable := TRUE;
   instcmSuctionPadTopRightVaccum.statProcessValues.referenceDesignator := WSTRING#'U1.EM2 SemiAutoSplice.cmSuctionPadTopRightVac';
   instcmSuctionPadTopRightVaccum.statProcessValues.commandHomePos := FALSE;
   instcmSuctionPadTopRightVaccum.statProcessValues.commandWorkPos := FALSE;
   instcmSuctionPadTopRightVaccum.statProcessValues.goToHomePos := FALSE;
   instcmSuctionPadTopRightVaccum.statProcessValues.goToWorkPos := FALSE;
   instcmSuctionPadTopRightVaccum.statProcessValues.inHomePos := TRUE;
   instcmSuctionPadTopRightVaccum.statProcessValues.inWorkPos := FALSE;
   instcmSuctionPadTopRightVaccum.statProcessValues.reset := FALSE;
   instcmSuctionPadTopRightVaccum.statProcessValues.enableManualCmds := TRUE;
   instcmSuctionPadTopRightVaccum.statProcessValues.error := FALSE;
   instcmSuctionPadTopRightVaccum.statProcessValues.interlockHomePos := TRUE;
   instcmSuctionPadTopRightVaccum.statProcessValues.interlockWorkPos := TRUE;
   instcmSuctionPadTopRightVaccum.statProcessValues.status := 16#7003;
   instcmSuctionPadTopRightVaccum.statProcessValues.interlockWarningWorkPos := FALSE;
   instcmSuctionPadTopRightVaccum.statProcessValues.interlockWarningHomePos := FALSE;
   instcmSuctionPadTopRightVaccum.statCurrentInputs.commandHomePos := FALSE;
   instcmSuctionPadTopRightVaccum.statCurrentInputs.commandWorkPos := FALSE;
   instcmSuctionPadTopRightVaccum.statCurrentInputs.reset := FALSE;
   instcmSuctionPadTopRightVaccum.statPreviousInputs.commandHomePos := FALSE;
   instcmSuctionPadTopRightVaccum.statPreviousInputs.commandWorkPos := FALSE;
   instcmSuctionPadTopRightVaccum.statPreviousInputs.reset := FALSE;
   instcmSuctionPadTopRightVaccum.statCurrentInterface.commandHomePos := FALSE;
   instcmSuctionPadTopRightVaccum.statCurrentInterface.commandWorkPos := FALSE;
   instcmSuctionPadTopRightVaccum.statCurrentInterface.reset := FALSE;
   instcmSuctionPadTopRightVaccum.statPreviousInterface.commandHomePos := FALSE;
   instcmSuctionPadTopRightVaccum.statPreviousInterface.commandWorkPos := FALSE;
   instcmSuctionPadTopRightVaccum.statPreviousInterface.reset := FALSE;
   instcmSuctionPadTopRightVaccum.statEmptyDiagnostics.status := 16#0000;
   instcmSuctionPadTopRightVaccum.statEmptyDiagnostics.subfunctionStatus := 16#0000;
   instcmSuctionPadTopRightVaccum.statEmptyDiagnostics.stateNumber := 0;
   instcmSuctionPadTopRightVaccum.instTimerReachPos.PT := T#0MS;
   instcmSuctionPadTopRightVaccum.instTimerReachPos.IN := FALSE;
   instcmSuctionPadTopRightVaccum.instTimerLeavePos.PT := T#0MS;
   instcmSuctionPadTopRightVaccum.instTimerLeavePos.IN := FALSE;
   instcmSuctionPadTopRightVaccum.instTimerDiscrepancyCheck.PT := T#0MS;
   instcmSuctionPadTopRightVaccum.instTimerDiscrepancyCheck.IN := FALSE;
   instcmSuctionPadTopRightVaccum.statDisableAlarms := FALSE;
   instcmSuctionPadTopRightVaccum.statDiagnostics.status := 16#7003;
   instcmSuctionPadTopRightVaccum.statDiagnostics.subfunctionStatus := 16#0000;
   instcmSuctionPadTopRightVaccum.statDiagnostics.stateNumber := 0;
   instcmSuctionPadTopRightVaccum.statEnablePrevious := TRUE;
   instcmSuctionPadTopRightVaccum.statFirstCall := FALSE;
   instcmSuctionPadTopRightVaccum.statResetPrevious := FALSE;
   instcmSuctionPadTopRightVaccum.statValid := TRUE;
   instcmSuctionPadTopRightVaccum.statBusy := TRUE;
   instcmSuctionPadTopRightVaccum.statError := FALSE;
   instcmSuctionPadTopRightVaccum.statInterlockWorkOff := FALSE;
   instcmSuctionPadTopRightVaccum.statInterlockHomeOff := FALSE;
   instcmSuctionPadTopRightVaccum.statFbState := 50;
   instcmSuctionPadTopRightVaccum.statFbStatePrevious := 50;
   instcmSuctionPadTopRightVaccum.statErrorUserCleared := FALSE;
   instcmSuctionPadTopRightVaccum.statErrorAutoCleared := FALSE;
   instcmSuctionPadTopRightVaccum.statErrorState := 16#0000;
   instcmSuctionPadTopRightVaccum.statDisablingCompleted := FALSE;
   instcmSuctionPadTopRightVaccum.statFeedbackHomePos := TRUE;
   instcmSuctionPadTopRightVaccum.statFeedbackWorkPos := FALSE;
   instCmSuctionPadBtmLeftVaccum.enable := TRUE;
   instCmSuctionPadBtmLeftVaccum.parentReferenceDesignator := WSTRING#'U1.EM2 SemiAutoSplice';
   instCmSuctionPadBtmLeftVaccum.feedbackHomePos := TRUE;
   instCmSuctionPadBtmLeftVaccum.feedbackWorkPos := FALSE;
   instCmSuctionPadBtmLeftVaccum.enableManualCmds := TRUE;
   instCmSuctionPadBtmLeftVaccum.interlockWorkPos := TRUE;
   instCmSuctionPadBtmLeftVaccum.interlockHomePos := TRUE;
   instCmSuctionPadBtmLeftVaccum.goToHomePos := FALSE;
   instCmSuctionPadBtmLeftVaccum.goToWorkPos := FALSE;
   instCmSuctionPadBtmLeftVaccum.statProcessValues.enable := TRUE;
   instCmSuctionPadBtmLeftVaccum.statProcessValues.referenceDesignator := WSTRING#'U1.EM2 SemiAutoSplice.cmSuctionPadBtmLeftVac';
   instCmSuctionPadBtmLeftVaccum.statProcessValues.commandHomePos := FALSE;
   instCmSuctionPadBtmLeftVaccum.statProcessValues.commandWorkPos := FALSE;
   instCmSuctionPadBtmLeftVaccum.statProcessValues.goToHomePos := FALSE;
   instCmSuctionPadBtmLeftVaccum.statProcessValues.goToWorkPos := FALSE;
   instCmSuctionPadBtmLeftVaccum.statProcessValues.inHomePos := TRUE;
   instCmSuctionPadBtmLeftVaccum.statProcessValues.inWorkPos := FALSE;
   instCmSuctionPadBtmLeftVaccum.statProcessValues.reset := FALSE;
   instCmSuctionPadBtmLeftVaccum.statProcessValues.enableManualCmds := TRUE;
   instCmSuctionPadBtmLeftVaccum.statProcessValues.error := FALSE;
   instCmSuctionPadBtmLeftVaccum.statProcessValues.interlockHomePos := TRUE;
   instCmSuctionPadBtmLeftVaccum.statProcessValues.interlockWorkPos := TRUE;
   instCmSuctionPadBtmLeftVaccum.statProcessValues.status := 16#7003;
   instCmSuctionPadBtmLeftVaccum.statProcessValues.interlockWarningWorkPos := FALSE;
   instCmSuctionPadBtmLeftVaccum.statProcessValues.interlockWarningHomePos := FALSE;
   instCmSuctionPadBtmLeftVaccum.statCurrentInputs.commandHomePos := FALSE;
   instCmSuctionPadBtmLeftVaccum.statCurrentInputs.commandWorkPos := FALSE;
   instCmSuctionPadBtmLeftVaccum.statCurrentInputs.reset := FALSE;
   instCmSuctionPadBtmLeftVaccum.statPreviousInputs.commandHomePos := FALSE;
   instCmSuctionPadBtmLeftVaccum.statPreviousInputs.commandWorkPos := FALSE;
   instCmSuctionPadBtmLeftVaccum.statPreviousInputs.reset := FALSE;
   instCmSuctionPadBtmLeftVaccum.statCurrentInterface.commandHomePos := FALSE;
   instCmSuctionPadBtmLeftVaccum.statCurrentInterface.commandWorkPos := FALSE;
   instCmSuctionPadBtmLeftVaccum.statCurrentInterface.reset := FALSE;
   instCmSuctionPadBtmLeftVaccum.statPreviousInterface.commandHomePos := FALSE;
   instCmSuctionPadBtmLeftVaccum.statPreviousInterface.commandWorkPos := FALSE;
   instCmSuctionPadBtmLeftVaccum.statPreviousInterface.reset := FALSE;
   instCmSuctionPadBtmLeftVaccum.statEmptyDiagnostics.status := 16#0000;
   instCmSuctionPadBtmLeftVaccum.statEmptyDiagnostics.subfunctionStatus := 16#0000;
   instCmSuctionPadBtmLeftVaccum.statEmptyDiagnostics.stateNumber := 0;
   instCmSuctionPadBtmLeftVaccum.instTimerReachPos.PT := T#0MS;
   instCmSuctionPadBtmLeftVaccum.instTimerReachPos.IN := FALSE;
   instCmSuctionPadBtmLeftVaccum.instTimerLeavePos.PT := T#0MS;
   instCmSuctionPadBtmLeftVaccum.instTimerLeavePos.IN := FALSE;
   instCmSuctionPadBtmLeftVaccum.instTimerDiscrepancyCheck.PT := T#0MS;
   instCmSuctionPadBtmLeftVaccum.instTimerDiscrepancyCheck.IN := FALSE;
   instCmSuctionPadBtmLeftVaccum.statDisableAlarms := FALSE;
   instCmSuctionPadBtmLeftVaccum.statDiagnostics.status := 16#7003;
   instCmSuctionPadBtmLeftVaccum.statDiagnostics.subfunctionStatus := 16#0000;
   instCmSuctionPadBtmLeftVaccum.statDiagnostics.stateNumber := 0;
   instCmSuctionPadBtmLeftVaccum.statEnablePrevious := TRUE;
   instCmSuctionPadBtmLeftVaccum.statFirstCall := FALSE;
   instCmSuctionPadBtmLeftVaccum.statResetPrevious := FALSE;
   instCmSuctionPadBtmLeftVaccum.statValid := TRUE;
   instCmSuctionPadBtmLeftVaccum.statBusy := TRUE;
   instCmSuctionPadBtmLeftVaccum.statError := FALSE;
   instCmSuctionPadBtmLeftVaccum.statInterlockWorkOff := FALSE;
   instCmSuctionPadBtmLeftVaccum.statInterlockHomeOff := FALSE;
   instCmSuctionPadBtmLeftVaccum.statFbState := 50;
   instCmSuctionPadBtmLeftVaccum.statFbStatePrevious := 50;
   instCmSuctionPadBtmLeftVaccum.statErrorUserCleared := FALSE;
   instCmSuctionPadBtmLeftVaccum.statErrorAutoCleared := FALSE;
   instCmSuctionPadBtmLeftVaccum.statErrorState := 16#0000;
   instCmSuctionPadBtmLeftVaccum.statDisablingCompleted := FALSE;
   instCmSuctionPadBtmLeftVaccum.statFeedbackHomePos := TRUE;
   instCmSuctionPadBtmLeftVaccum.statFeedbackWorkPos := FALSE;
   instCmSuctionPadBtmRightVaccum.enable := TRUE;
   instCmSuctionPadBtmRightVaccum.parentReferenceDesignator := WSTRING#'U1.EM2 SemiAutoSplice';
   instCmSuctionPadBtmRightVaccum.feedbackHomePos := TRUE;
   instCmSuctionPadBtmRightVaccum.feedbackWorkPos := FALSE;
   instCmSuctionPadBtmRightVaccum.enableManualCmds := TRUE;
   instCmSuctionPadBtmRightVaccum.interlockWorkPos := TRUE;
   instCmSuctionPadBtmRightVaccum.interlockHomePos := TRUE;
   instCmSuctionPadBtmRightVaccum.goToHomePos := FALSE;
   instCmSuctionPadBtmRightVaccum.goToWorkPos := FALSE;
   instCmSuctionPadBtmRightVaccum.statProcessValues.enable := TRUE;
   instCmSuctionPadBtmRightVaccum.statProcessValues.referenceDesignator := WSTRING#'U1.EM2 SemiAutoSplice.cmSuctionPadBtmRightVac';
   instCmSuctionPadBtmRightVaccum.statProcessValues.commandHomePos := FALSE;
   instCmSuctionPadBtmRightVaccum.statProcessValues.commandWorkPos := FALSE;
   instCmSuctionPadBtmRightVaccum.statProcessValues.goToHomePos := FALSE;
   instCmSuctionPadBtmRightVaccum.statProcessValues.goToWorkPos := FALSE;
   instCmSuctionPadBtmRightVaccum.statProcessValues.inHomePos := TRUE;
   instCmSuctionPadBtmRightVaccum.statProcessValues.inWorkPos := FALSE;
   instCmSuctionPadBtmRightVaccum.statProcessValues.reset := FALSE;
   instCmSuctionPadBtmRightVaccum.statProcessValues.enableManualCmds := TRUE;
   instCmSuctionPadBtmRightVaccum.statProcessValues.error := FALSE;
   instCmSuctionPadBtmRightVaccum.statProcessValues.interlockHomePos := TRUE;
   instCmSuctionPadBtmRightVaccum.statProcessValues.interlockWorkPos := TRUE;
   instCmSuctionPadBtmRightVaccum.statProcessValues.status := 16#7003;
   instCmSuctionPadBtmRightVaccum.statProcessValues.interlockWarningWorkPos := FALSE;
   instCmSuctionPadBtmRightVaccum.statProcessValues.interlockWarningHomePos := FALSE;
   instCmSuctionPadBtmRightVaccum.statCurrentInputs.commandHomePos := FALSE;
   instCmSuctionPadBtmRightVaccum.statCurrentInputs.commandWorkPos := FALSE;
   instCmSuctionPadBtmRightVaccum.statCurrentInputs.reset := FALSE;
   instCmSuctionPadBtmRightVaccum.statPreviousInputs.commandHomePos := FALSE;
   instCmSuctionPadBtmRightVaccum.statPreviousInputs.commandWorkPos := FALSE;
   instCmSuctionPadBtmRightVaccum.statPreviousInputs.reset := FALSE;
   instCmSuctionPadBtmRightVaccum.statCurrentInterface.commandHomePos := FALSE;
   instCmSuctionPadBtmRightVaccum.statCurrentInterface.commandWorkPos := FALSE;
   instCmSuctionPadBtmRightVaccum.statCurrentInterface.reset := FALSE;
   instCmSuctionPadBtmRightVaccum.statPreviousInterface.commandHomePos := FALSE;
   instCmSuctionPadBtmRightVaccum.statPreviousInterface.commandWorkPos := FALSE;
   instCmSuctionPadBtmRightVaccum.statPreviousInterface.reset := FALSE;
   instCmSuctionPadBtmRightVaccum.statEmptyDiagnostics.status := 16#0000;
   instCmSuctionPadBtmRightVaccum.statEmptyDiagnostics.subfunctionStatus := 16#0000;
   instCmSuctionPadBtmRightVaccum.statEmptyDiagnostics.stateNumber := 0;
   instCmSuctionPadBtmRightVaccum.instTimerReachPos.PT := T#0MS;
   instCmSuctionPadBtmRightVaccum.instTimerReachPos.IN := FALSE;
   instCmSuctionPadBtmRightVaccum.instTimerLeavePos.PT := T#0MS;
   instCmSuctionPadBtmRightVaccum.instTimerLeavePos.IN := FALSE;
   instCmSuctionPadBtmRightVaccum.instTimerDiscrepancyCheck.PT := T#0MS;
   instCmSuctionPadBtmRightVaccum.instTimerDiscrepancyCheck.IN := FALSE;
   instCmSuctionPadBtmRightVaccum.statDisableAlarms := FALSE;
   instCmSuctionPadBtmRightVaccum.statDiagnostics.status := 16#7003;
   instCmSuctionPadBtmRightVaccum.statDiagnostics.subfunctionStatus := 16#0000;
   instCmSuctionPadBtmRightVaccum.statDiagnostics.stateNumber := 0;
   instCmSuctionPadBtmRightVaccum.statEnablePrevious := TRUE;
   instCmSuctionPadBtmRightVaccum.statFirstCall := FALSE;
   instCmSuctionPadBtmRightVaccum.statResetPrevious := FALSE;
   instCmSuctionPadBtmRightVaccum.statValid := TRUE;
   instCmSuctionPadBtmRightVaccum.statBusy := TRUE;
   instCmSuctionPadBtmRightVaccum.statError := FALSE;
   instCmSuctionPadBtmRightVaccum.statInterlockWorkOff := FALSE;
   instCmSuctionPadBtmRightVaccum.statInterlockHomeOff := FALSE;
   instCmSuctionPadBtmRightVaccum.statFbState := 50;
   instCmSuctionPadBtmRightVaccum.statFbStatePrevious := 50;
   instCmSuctionPadBtmRightVaccum.statErrorUserCleared := FALSE;
   instCmSuctionPadBtmRightVaccum.statErrorAutoCleared := FALSE;
   instCmSuctionPadBtmRightVaccum.statErrorState := 16#0000;
   instCmSuctionPadBtmRightVaccum.statDisablingCompleted := FALSE;
   instCmSuctionPadBtmRightVaccum.statFeedbackHomePos := TRUE;
   instCmSuctionPadBtmRightVaccum.statFeedbackWorkPos := FALSE;
   instCmSuctionPadTopTapeVaccum.enable := TRUE;
   instCmSuctionPadTopTapeVaccum.parentReferenceDesignator := WSTRING#'U1.EM2 SemiAutoSplice';
   instCmSuctionPadTopTapeVaccum.feedbackHomePos := TRUE;
   instCmSuctionPadTopTapeVaccum.feedbackWorkPos := FALSE;
   instCmSuctionPadTopTapeVaccum.enableManualCmds := TRUE;
   instCmSuctionPadTopTapeVaccum.interlockWorkPos := TRUE;
   instCmSuctionPadTopTapeVaccum.interlockHomePos := TRUE;
   instCmSuctionPadTopTapeVaccum.goToHomePos := FALSE;
   instCmSuctionPadTopTapeVaccum.goToWorkPos := FALSE;
   instCmSuctionPadTopTapeVaccum.statProcessValues.enable := TRUE;
   instCmSuctionPadTopTapeVaccum.statProcessValues.referenceDesignator := WSTRING#'U1.EM2 SemiAutoSplice.cmSuctionPadTopTapeVac';
   instCmSuctionPadTopTapeVaccum.statProcessValues.commandHomePos := FALSE;
   instCmSuctionPadTopTapeVaccum.statProcessValues.commandWorkPos := FALSE;
   instCmSuctionPadTopTapeVaccum.statProcessValues.goToHomePos := FALSE;
   instCmSuctionPadTopTapeVaccum.statProcessValues.goToWorkPos := FALSE;
   instCmSuctionPadTopTapeVaccum.statProcessValues.inHomePos := TRUE;
   instCmSuctionPadTopTapeVaccum.statProcessValues.inWorkPos := FALSE;
   instCmSuctionPadTopTapeVaccum.statProcessValues.reset := FALSE;
   instCmSuctionPadTopTapeVaccum.statProcessValues.enableManualCmds := TRUE;
   instCmSuctionPadTopTapeVaccum.statProcessValues.error := FALSE;
   instCmSuctionPadTopTapeVaccum.statProcessValues.interlockHomePos := TRUE;
   instCmSuctionPadTopTapeVaccum.statProcessValues.interlockWorkPos := TRUE;
   instCmSuctionPadTopTapeVaccum.statProcessValues.status := 16#7003;
   instCmSuctionPadTopTapeVaccum.statProcessValues.interlockWarningWorkPos := FALSE;
   instCmSuctionPadTopTapeVaccum.statProcessValues.interlockWarningHomePos := FALSE;
   instCmSuctionPadTopTapeVaccum.statCurrentInputs.commandHomePos := FALSE;
   instCmSuctionPadTopTapeVaccum.statCurrentInputs.commandWorkPos := FALSE;
   instCmSuctionPadTopTapeVaccum.statCurrentInputs.reset := FALSE;
   instCmSuctionPadTopTapeVaccum.statPreviousInputs.commandHomePos := FALSE;
   instCmSuctionPadTopTapeVaccum.statPreviousInputs.commandWorkPos := FALSE;
   instCmSuctionPadTopTapeVaccum.statPreviousInputs.reset := FALSE;
   instCmSuctionPadTopTapeVaccum.statCurrentInterface.commandHomePos := FALSE;
   instCmSuctionPadTopTapeVaccum.statCurrentInterface.commandWorkPos := FALSE;
   instCmSuctionPadTopTapeVaccum.statCurrentInterface.reset := FALSE;
   instCmSuctionPadTopTapeVaccum.statPreviousInterface.commandHomePos := FALSE;
   instCmSuctionPadTopTapeVaccum.statPreviousInterface.commandWorkPos := FALSE;
   instCmSuctionPadTopTapeVaccum.statPreviousInterface.reset := FALSE;
   instCmSuctionPadTopTapeVaccum.statEmptyDiagnostics.status := 16#0000;
   instCmSuctionPadTopTapeVaccum.statEmptyDiagnostics.subfunctionStatus := 16#0000;
   instCmSuctionPadTopTapeVaccum.statEmptyDiagnostics.stateNumber := 0;
   instCmSuctionPadTopTapeVaccum.instTimerReachPos.PT := T#0MS;
   instCmSuctionPadTopTapeVaccum.instTimerReachPos.IN := FALSE;
   instCmSuctionPadTopTapeVaccum.instTimerLeavePos.PT := T#0MS;
   instCmSuctionPadTopTapeVaccum.instTimerLeavePos.IN := FALSE;
   instCmSuctionPadTopTapeVaccum.instTimerDiscrepancyCheck.PT := T#0MS;
   instCmSuctionPadTopTapeVaccum.instTimerDiscrepancyCheck.IN := FALSE;
   instCmSuctionPadTopTapeVaccum.statDisableAlarms := FALSE;
   instCmSuctionPadTopTapeVaccum.statDiagnostics.status := 16#7003;
   instCmSuctionPadTopTapeVaccum.statDiagnostics.subfunctionStatus := 16#0000;
   instCmSuctionPadTopTapeVaccum.statDiagnostics.stateNumber := 0;
   instCmSuctionPadTopTapeVaccum.statEnablePrevious := TRUE;
   instCmSuctionPadTopTapeVaccum.statFirstCall := FALSE;
   instCmSuctionPadTopTapeVaccum.statResetPrevious := FALSE;
   instCmSuctionPadTopTapeVaccum.statValid := TRUE;
   instCmSuctionPadTopTapeVaccum.statBusy := TRUE;
   instCmSuctionPadTopTapeVaccum.statError := FALSE;
   instCmSuctionPadTopTapeVaccum.statInterlockWorkOff := FALSE;
   instCmSuctionPadTopTapeVaccum.statInterlockHomeOff := FALSE;
   instCmSuctionPadTopTapeVaccum.statFbState := 50;
   instCmSuctionPadTopTapeVaccum.statFbStatePrevious := 50;
   instCmSuctionPadTopTapeVaccum.statErrorUserCleared := FALSE;
   instCmSuctionPadTopTapeVaccum.statErrorAutoCleared := FALSE;
   instCmSuctionPadTopTapeVaccum.statErrorState := 16#0000;
   instCmSuctionPadTopTapeVaccum.statDisablingCompleted := FALSE;
   instCmSuctionPadTopTapeVaccum.statFeedbackHomePos := TRUE;
   instCmSuctionPadTopTapeVaccum.statFeedbackWorkPos := FALSE;
   instCmSuctionPadBtmTapeVaccum.enable := TRUE;
   instCmSuctionPadBtmTapeVaccum.parentReferenceDesignator := WSTRING#'U1.EM2 SemiAutoSplice';
   instCmSuctionPadBtmTapeVaccum.feedbackHomePos := TRUE;
   instCmSuctionPadBtmTapeVaccum.feedbackWorkPos := FALSE;
   instCmSuctionPadBtmTapeVaccum.enableManualCmds := TRUE;
   instCmSuctionPadBtmTapeVaccum.interlockWorkPos := TRUE;
   instCmSuctionPadBtmTapeVaccum.interlockHomePos := TRUE;
   instCmSuctionPadBtmTapeVaccum.goToHomePos := FALSE;
   instCmSuctionPadBtmTapeVaccum.goToWorkPos := FALSE;
   instCmSuctionPadBtmTapeVaccum.statProcessValues.enable := TRUE;
   instCmSuctionPadBtmTapeVaccum.statProcessValues.referenceDesignator := WSTRING#'U1.EM2 SemiAutoSplice.cmSuctionPadBtmTapeVac';
   instCmSuctionPadBtmTapeVaccum.statProcessValues.commandHomePos := FALSE;
   instCmSuctionPadBtmTapeVaccum.statProcessValues.commandWorkPos := FALSE;
   instCmSuctionPadBtmTapeVaccum.statProcessValues.goToHomePos := FALSE;
   instCmSuctionPadBtmTapeVaccum.statProcessValues.goToWorkPos := FALSE;
   instCmSuctionPadBtmTapeVaccum.statProcessValues.inHomePos := TRUE;
   instCmSuctionPadBtmTapeVaccum.statProcessValues.inWorkPos := FALSE;
   instCmSuctionPadBtmTapeVaccum.statProcessValues.reset := FALSE;
   instCmSuctionPadBtmTapeVaccum.statProcessValues.enableManualCmds := TRUE;
   instCmSuctionPadBtmTapeVaccum.statProcessValues.error := FALSE;
   instCmSuctionPadBtmTapeVaccum.statProcessValues.interlockHomePos := TRUE;
   instCmSuctionPadBtmTapeVaccum.statProcessValues.interlockWorkPos := TRUE;
   instCmSuctionPadBtmTapeVaccum.statProcessValues.status := 16#7003;
   instCmSuctionPadBtmTapeVaccum.statProcessValues.interlockWarningWorkPos := FALSE;
   instCmSuctionPadBtmTapeVaccum.statProcessValues.interlockWarningHomePos := FALSE;
   instCmSuctionPadBtmTapeVaccum.statCurrentInputs.commandHomePos := FALSE;
   instCmSuctionPadBtmTapeVaccum.statCurrentInputs.commandWorkPos := FALSE;
   instCmSuctionPadBtmTapeVaccum.statCurrentInputs.reset := FALSE;
   instCmSuctionPadBtmTapeVaccum.statPreviousInputs.commandHomePos := FALSE;
   instCmSuctionPadBtmTapeVaccum.statPreviousInputs.commandWorkPos := FALSE;
   instCmSuctionPadBtmTapeVaccum.statPreviousInputs.reset := FALSE;
   instCmSuctionPadBtmTapeVaccum.statCurrentInterface.commandHomePos := FALSE;
   instCmSuctionPadBtmTapeVaccum.statCurrentInterface.commandWorkPos := FALSE;
   instCmSuctionPadBtmTapeVaccum.statCurrentInterface.reset := FALSE;
   instCmSuctionPadBtmTapeVaccum.statPreviousInterface.commandHomePos := FALSE;
   instCmSuctionPadBtmTapeVaccum.statPreviousInterface.commandWorkPos := FALSE;
   instCmSuctionPadBtmTapeVaccum.statPreviousInterface.reset := FALSE;
   instCmSuctionPadBtmTapeVaccum.statEmptyDiagnostics.status := 16#0000;
   instCmSuctionPadBtmTapeVaccum.statEmptyDiagnostics.subfunctionStatus := 16#0000;
   instCmSuctionPadBtmTapeVaccum.statEmptyDiagnostics.stateNumber := 0;
   instCmSuctionPadBtmTapeVaccum.instTimerReachPos.PT := T#0MS;
   instCmSuctionPadBtmTapeVaccum.instTimerReachPos.IN := FALSE;
   instCmSuctionPadBtmTapeVaccum.instTimerLeavePos.PT := T#0MS;
   instCmSuctionPadBtmTapeVaccum.instTimerLeavePos.IN := FALSE;
   instCmSuctionPadBtmTapeVaccum.instTimerDiscrepancyCheck.PT := T#0MS;
   instCmSuctionPadBtmTapeVaccum.instTimerDiscrepancyCheck.IN := FALSE;
   instCmSuctionPadBtmTapeVaccum.statDisableAlarms := FALSE;
   instCmSuctionPadBtmTapeVaccum.statDiagnostics.status := 16#7003;
   instCmSuctionPadBtmTapeVaccum.statDiagnostics.subfunctionStatus := 16#0000;
   instCmSuctionPadBtmTapeVaccum.statDiagnostics.stateNumber := 0;
   instCmSuctionPadBtmTapeVaccum.statEnablePrevious := TRUE;
   instCmSuctionPadBtmTapeVaccum.statFirstCall := FALSE;
   instCmSuctionPadBtmTapeVaccum.statResetPrevious := FALSE;
   instCmSuctionPadBtmTapeVaccum.statValid := TRUE;
   instCmSuctionPadBtmTapeVaccum.statBusy := TRUE;
   instCmSuctionPadBtmTapeVaccum.statError := FALSE;
   instCmSuctionPadBtmTapeVaccum.statInterlockWorkOff := FALSE;
   instCmSuctionPadBtmTapeVaccum.statInterlockHomeOff := FALSE;
   instCmSuctionPadBtmTapeVaccum.statFbState := 50;
   instCmSuctionPadBtmTapeVaccum.statFbStatePrevious := 50;
   instCmSuctionPadBtmTapeVaccum.statErrorUserCleared := FALSE;
   instCmSuctionPadBtmTapeVaccum.statErrorAutoCleared := FALSE;
   instCmSuctionPadBtmTapeVaccum.statErrorState := 16#0000;
   instCmSuctionPadBtmTapeVaccum.statDisablingCompleted := FALSE;
   instCmSuctionPadBtmTapeVaccum.statFeedbackHomePos := TRUE;
   instCmSuctionPadBtmTapeVaccum.statFeedbackWorkPos := FALSE;
   instManageAlarms.proDiagState.Total_Number := 448;
   instManageAlarms.proDiagState.All := FALSE;
   instManageAlarms.proDiagState.O := FALSE;
   instManageAlarms.proDiagState.I := FALSE;
   instManageAlarms.proDiagState.R := FALSE;
   instManageAlarms.proDiagState."A" := FALSE;
   instManageAlarms.proDiagState.P := FALSE;
   instManageAlarms.proDiagState.Merr := FALSE;
   instManageAlarms.proDiagState.Mtxt := FALSE;
   instManageAlarms.proDiagState.SV_Types := 16#00;
   instManageAlarms.proDiagState.C1 := FALSE;
   instManageAlarms.proDiagState.C2 := FALSE;
   instManageAlarms.proDiagState.C3 := FALSE;
   instManageAlarms.proDiagState.C4 := FALSE;
   instManageAlarms.proDiagState.C5 := FALSE;
   instManageAlarms.proDiagState.C6 := FALSE;
   instManageAlarms.proDiagState.C7 := FALSE;
   instManageAlarms.proDiagState.C8 := FALSE;
   instManageAlarms.proDiagState.Categories := 16#00;
   instManageAlarms.proDiagState.Sub_Cat_1 := 16#0000_0000;
   instManageAlarms.proDiagState.Sub_Cat_2 := 16#0000_0000;
   instManageAlarms.proDiagState.Reserved := 16#00;
   instManageAlarms.parentAlarmDB.error := FALSE;
   instManageAlarms.parentAlarmDB.warning := FALSE;
   instManageAlarms.parentAlarmDB.info := FALSE;
   instManageAlarms.alarmDB.error := FALSE;
   instManageAlarms.alarmDB.warning := FALSE;
   instManageAlarms.alarmDB.info := FALSE;
   instManageAlarms.hmiInterfaceDB.error := FALSE;
   instManageAlarms.hmiInterfaceDB.warning := FALSE;
   instManageAlarms.hmiInterfaceDB.info := FALSE;
   statUnitStatus.acknowledgeActive := FALSE;
   statUnitStatus.alarmsDisabled := FALSE;
   statUnitStatus.simulationActive := FALSE;
   statUnitStatus.safetyReleased := TRUE;
   statUnitStatus.state.current := 2;
   statUnitStatus.state.clearing := FALSE;
   statUnitStatus.state.stopped := TRUE;
   statUnitStatus.state.starting := FALSE;
   statUnitStatus.state.idle := FALSE;
   statUnitStatus.state.suspended := FALSE;
   statUnitStatus.state.execute := FALSE;
   statUnitStatus.state.stopping := FALSE;
   statUnitStatus.state.aborting := FALSE;
   statUnitStatus.state.aborted := FALSE;
   statUnitStatus.state.holding := FALSE;
   statUnitStatus.state.held := FALSE;
   statUnitStatus.state.unholding := FALSE;
   statUnitStatus.state.suspending := FALSE;
   statUnitStatus.state.unsuspending := FALSE;
   statUnitStatus.state.resetting := FALSE;
   statUnitStatus.state.completing := FALSE;
   statUnitStatus.state.complete := FALSE;
END_DATA_BLOCK
